//{attribute 'qualified_only'}
VAR_GLOBAL
	Pendulum : Pendulum4Tc;
END_VAR

(* stored: Version 1.1.0.1, ProductVersion 3.1.4024.12
   GVL GVLPendulum: Id {cabe1232-263f-4474-a80c-149b745e081a} *)
